// TIA Portal V18 export
DATA_BLOCK "AHUEqp"   // DB104
{ S7_Optimized_Access := 'FALSE' }
VERSION : 0.1
// stored: AutoNumber false, DBAccessibleFromOPCUA true, IsOnlyStoredInLoadMemory false, IsWriteProtectedInAS false
   VAR RETAIN
      Eqp { S7_SetPoint := 'True'} : "UDT_AHUEqp";
   END_VAR
BEGIN
   Eqp.Cfg.cFan[1] := 4;
   Eqp.Cfg.cFan[2] := 3;
   Eqp.Cfg.cExtractDumper[1] := 2;
   Eqp.Cfg.cMixingDumper[1..2] := 2;
   Eqp.Cfg.cHeater[1..2] := 2;
   Eqp.LimiterGridOperation.rFan[1..3] := 1.0;
   Eqp.LimiterGridOperation.rExtractDumper[1..3] := 1.0;
   Eqp.LimiterGridOperation.rMixingDumper[1..3] := 1.0;
   Eqp.LimiterGridOperation.rHeater[1..3] := 1.0;
   Eqp.LimiterGridOperation.rCooler[1..3] := 1.0;
   Eqp.LimiterGridOperation.rWHU[1..3] := 1.0;
   Eqp.LimiterDieselOperation.rFan[1..3] := 0.5;
   Eqp.LimiterDieselOperation.rExtractDumper[1..3] := 0.5;
   Eqp.LimiterDieselOperation.rMixingDumper[1..3] := 0.5;
   Eqp.LimiterDieselOperation.rHeater[1..3] := 1.0;
   Eqp.LimiterDieselOperation.rCooler[1..3] := 0.5;
   Eqp.LimiterDieselOperation.rWHU[1..3] := 1.0;
END_DATA_BLOCK
